FUNCTION_BLOCK FB_ZAxisRef EXTENDS FB_HwModule
VAR_INPUT
	stInput 			: ST_ZAxisRef_In;
	stOutput 			: ST_ZAxisRef_Out;
	stStatus			: ST_ZAxisStatus;
	
	eDetectedToolType 	: E_MzToolType; //Sdo , wird nur bei Kopfbasisplatinen mir Toolerkennung benutzt und wird bei 
										//A_PrepareAxis in FB_MultiZRef ausgelesen
	eFixedToolType		: E_MzToolType; //Sdo, wird in den Objekten gesetzt und dann in A_SetConfig oder A_SetConfigLegacy
										//in FB_MultiZRef ausgelesen 
	
	bHasTool	: BOOL;
	sTmcVersion	: STRING(5);
	nTmcModulId	: UINT;
	nToolVersion: USINT;
	bIsSubAxis	: BOOL; //Ist eine Unterachse z.B. vom Stempel (wird vom Stempel gesteuert)
	bIngoreError: BOOL; //verhindert das Abfangen eines Fehlers in "A_Monitor"
	pCurrentFb	: POINTER TO PVOID;
END_VAR

VAR_OUTPUT
	pMultiZRef : POINTER TO FB_MultiZRef;
	nChannel : USINT;
END_VAR

VAR PERSISTENT
	rMaxSpeed 		: REAL;
	rRefPos 		: REAL;
	rMaxPos			: REAL;
	rMinPos			: REAL;
	rHomePos		: REAL;
	rAxisLength		: REAL;
	rSliderLength	: REAL;
	bInvertInitDir	: BOOL;
END_VAR

VAR
	nZSensorID  : DINT;
END_VAR

METHOD FB_init : BOOL
VAR_INPUT
	bInitRetains : BOOL; // if TRUE, the retain variables are initialized (warm start / cold start)
	bInCopyCode : BOOL;  // if TRUE, the instance afterwards gets moved into the copy code (online change)
	pMultiZRef : POINTER TO FB_MultiZRef;
END_VAR

VAR
	nFirstAdress : PVOID;
	nSelfAdress : PVOID;
END_VAR
THIS^.pMultiZRef := pMultiZRef;
nFirstAdress := ADR(pMultiZRef^.aFbZAxisRef);
nSelfAdress := THIS;
{IF hasvalue (RegisterSize, '32')}
nChannel := UDINT_TO_USINT((nSelfAdress - nFirstAdress)/SIZEOF(THIS^) + 1);
{ELSE}
nChannel := ULINT_TO_USINT((nSelfAdress - nFirstAdress)/SIZEOF(THIS^) + 1);
{END_IF}
stHardwareId.eGroup := E_HardwareGrp.AxisZ;
stHardwareId.nItem := nChannel;
END_METHOD

METHOD M_GetHwInfo : ST_HardwareInfo
VAR_INPUT
END_VAR
M_GetHwInfo := SUPER^.M_GetHwInfo();
M_GetHwInfo.sHardwVersion := UINT_TO_STRING(nTmcModulId);
M_GetHwInfo.sSoftwVersion := sTmcVersion;
M_GetHwInfo.sSoftwVersion2 := USINT_TO_STRING(nToolVersion);
END_METHOD

METHOD M_RenewHwId
VAR_INPUT
END_VAR

VAR
	stHwIdParent : ST_HardwareId;
END_VAR
stHwIdParent := pMultiZRef^.P_stHardwareId;
stHardwareId.nParentItem := stHwIdParent.nItem;
END_METHOD

PROPERTY P_bInvertInitDir : BOOL
GET
P_bInvertInitDir := bInvertInitDir;
END_GET
SET
bInvertInitDir := P_bInvertInitDir;
fbSettings.M_WritePersData();
END_SET
END_PROPERTY

PROPERTY P_nZSensorID : DINT
GET
P_nZSensorID := nZSensorID;
END_GET
SET
nZSensorID := P_nZSensorID;
END_SET
END_PROPERTY

PROPERTY P_rAbsTargetPos : REAL
SET
stOutput.nTrgtPos := REAL_TO_DINT(rAxisLength - rSliderLength - P_rAbsTargetPos);
END_SET
END_PROPERTY

PROPERTY P_rAxisLength : REAL
GET
P_rAxisLength := rAxisLength;
END_GET
SET
rAxisLength := P_rAxisLength;
fbSettings.M_WritePersData();
END_SET
END_PROPERTY

PROPERTY P_rCurrentPos : REAL
GET
P_rCurrentPos := MIN(rAxisLength - rSliderLength - DINT_TO_REAL(stInput.nCurrentPos),rMaxPos);
END_GET
END_PROPERTY

PROPERTY P_rHomePos : REAL
GET
P_rHomePos := rHomePos;
END_GET
SET
rHomePos := P_rHomePos;
fbSettings.M_WritePersData();
END_SET
END_PROPERTY

PROPERTY P_rMaxPos : REAL
GET
P_rMaxPos := rMaxPos;
END_GET
SET
rMaxPos := P_rMaxPos;
END_SET
END_PROPERTY

PROPERTY P_rMaxSpeed : REAL
GET
P_rMaxSpeed := rMaxSpeed;
END_GET
SET
rMaxSpeed := P_rMaxSpeed;
fbSettings.M_WritePersData();
END_SET
END_PROPERTY

PROPERTY P_rMinPos : REAL
GET
P_rMinPos := rMinPos;
END_GET
SET
rMinPos := P_rMinPos;
fbSettings.M_WritePersData();
END_SET
END_PROPERTY

PROPERTY P_rRefPos : REAL
GET
P_rRefPos := rRefPos;
END_GET
SET
rRefPos := P_rRefPos;
fbSettings.M_WritePersData();
END_SET
END_PROPERTY

PROPERTY P_rRelTargetPos : REAL
SET
stOutput.nTrgtPos := REAL_TO_DINT(- P_rRelTargetPos);
END_SET
END_PROPERTY

PROPERTY P_rSliderLength : REAL
GET
P_rSliderLength := rSliderLength;
END_GET
SET
rSliderLength := P_rSliderLength;
fbSettings.M_WritePersData();
END_SET
END_PROPERTY

PROPERTY P_rSpeed : REAL
GET
END_GET
SET
END_SET
END_PROPERTY

END_FUNCTION_BLOCK

(* stored: Version 1.1.0.1, ProductVersion 3.1.4022.18
   POU FB_ZAxisRef: Id {fd9020f6-1dda-4da0-abca-7706599353b8}, SpecialFunc None
   Method FB_init: Id {eaecb542-800c-4386-9b17-3394eb31f6c1}
   Method M_GetHwInfo: Id {f55e5975-7bf2-454d-be80-41bb09486f0f}
   Method M_RenewHwId: Id {545992a0-d838-4acb-8411-721782728375}
   Property P_bInvertInitDir: Id {d735c89c-979e-4ee6-ac91-1c72563c0080}
   Get Get: Id {b38e17ef-ebbe-4450-8ca3-1a486c26f0be}
   Set Set: Id {134bf3ea-82af-4d08-8bbb-282b08969207}
   Property P_nZSensorID: Id {0e65d215-607e-4246-987c-9b62c4f53603}
   Get Get: Id {c24ac606-3599-46f8-977a-6b2229941e04}
   Set Set: Id {2d2a0d8e-1be8-422c-8630-2d911aed2217}
   Property P_rAbsTargetPos: Id {de0c2abf-58c4-4d7b-b245-36411b7b66ba}
   Set Set: Id {0cfeff5f-6c6f-44b1-b536-2252f9547489}
   Property P_rAxisLength: Id {535886d6-f7dc-433d-a1f7-3427a98403c7}
   Get Get: Id {8ef7dd5d-2e58-4273-829f-063dadda6457}
   Set Set: Id {e410fc68-a5a7-4fec-8ada-dd142b4f4651}
   Property P_rCurrentPos: Id {c9c91295-bd23-409d-961f-95411143990e}
   Get Get: Id {67130349-ccad-42e0-a1bd-db9c3d887585}
   Property P_rHomePos: Id {c4ca3150-806a-449b-a446-f0067796acec}
   Get Get: Id {2c28c3e9-1712-421a-8141-3da84b3a1274}
   Set Set: Id {9d25bc1b-5d87-40cc-8547-707ee1978478}
   Property P_rMaxPos: Id {fc2cf8e1-c1b0-42e1-ab9d-254065c30126}
   Get Get: Id {4b7efe2f-4750-4c6e-86fb-38e626163540}
   Set Set: Id {ff4b6452-b21c-48ff-a8f7-847b3c877a01}
   Property P_rMaxSpeed: Id {3aed17fb-2ddb-4115-bd78-e40a26dac211}
   Get Get: Id {a2c00309-594f-4a44-af55-7e19a09bd278}
   Set Set: Id {9b8c5e54-4591-480b-8e91-ab911892a00a}
   Property P_rMinPos: Id {9d668293-f955-48dd-85b8-10624b449367}
   Get Get: Id {4d60eba6-700e-47b8-9f91-a152701f772d}
   Set Set: Id {0fa1fa49-88c9-48ff-aea9-932719f07624}
   Property P_rRefPos: Id {27642a54-d99c-415f-b088-7259a2c20b08}
   Get Get: Id {422318f7-58d6-4c31-a11c-80d4d95b7fcc}
   Set Set: Id {b7b9eb0c-cd29-4cb0-8dd8-669446eb7221}
   Property P_rRelTargetPos: Id {24411efb-88f4-428e-8b74-83aa62b8f06b}
   Set Set: Id {f05fbc19-6466-4f1b-aa20-f1273f8cdc34}
   Property P_rSliderLength: Id {1c6e2f5f-e567-40c9-8132-817a509553cf}
   Get Get: Id {4cc4196f-71bc-4a07-8b40-05ad8f74b5da}
   Set Set: Id {dc99d5cc-57d5-484b-abca-1a5393a5bb0d}
   Property P_rSpeed: Id {b23d854b-ad79-4ed4-baf5-0b296cfdadd3}
   Get Get: Id {9602764d-7d8c-4a2f-bb8b-3eb8a25487db}
   Set Set: Id {2eca0eed-d2b0-40cb-960a-b591ea8b1f60} *)
